PROGRAM MAIN
VAR
	fbBlinklicht : FB_Blinklicht;
	fbVereinzelung : FB_Vereinzelung;
	fbezylinder1 : FB_EZylinder;
	fbezylinder2 : FB_EZylinder;
	fbAmpel : FB_Ampel;
	fbTransport : FB_Transport;
	fbDispenser : FB_Dispenser;
	fbAbfuellmodul : FB_Abfuellmodul;
	fbManAchseX : FB_ManAchse;
	fbManAchseY : FB_ManAchse;
	fbManAchseZ : FB_ManAchse;
	ix : UINT;
	ry : REAL;
	ax : Axis_Ref;
END_VAR

ry := FUN_SCALE(TO_REAL(ix),4096,0,350,0);

	
fbAbfuellmodul(
	bEnable:= IFC_HW.bEnable, 
	bExecute:= IFC_HW.bExecute, 
	nstation:= , 
	bEinzelSens1:= IFC_HW.bEinzelSens1, 
	bEinzelSens2:= IFC_HW.bEinzelSens2, 
	bEinzelSens3:= IFC_HW.bEinzelSens3, 
	bEinzelSens4:= IFC_HW.bBandSens1, 
	bBandSens1:= IFC_HW.bBandSens1, 
	bBandSens2:= IFC_HW.bBandSens2, 
	bBandSens3:= IFC_HW.bBandSens3, 
	bBandSens4:= IFC_HW.bBandSens4, 
	bstopper1=> IFC_HW.bBandHub1, 
	bstopper2=> IFC_HW.bBandHub2, 
	bstopper3=>IFC_HW.bBandHub3, 
	estate=> , 
	bgate1=> fbeZylinder1.bgate, 
	bgate2=> fbeZylinder2.bgate, 
	axTransport:= IFC_HW.ax_BandMotor, 
	axDisp1:= IFC_HW.ax_Extruder1, 
	axDisp2:= IFC_HW.ax_Extruder2, 
	axDisp3:= IFC_HW.ax_Extruder3);
	
(*				
fbVereinzelung(
	benable:= IFC_HW.bEnable, 
	bexecute:= IFC_HW.bExecute, 
	bsensor1:= IFC_HW.bEinzelSens1, 
	bsensor2:= IFC_HW.bEinzelSens2, 
	bsensor3:= IFC_HW.bEinzelSens3, 
	bsensor4:= IFC_HW.bBandsens1, 
	bgate1=> fbeZylinder1.bgate, 
	bgate2=> fbeZylinder2.bgate, 
	estate=> );
	*)
	
	fbezylinder1(bgate:= , berror:= , bR1=>IFC_HW.bR1AKT1 , bR2=>IFC_HW.br2AKT1 );
	
	fbezylinder2(bgate:= , berror:= , bR1=>IFC_HW.bR1AKT2 , bR2=> IFC_HW.bR2AKT2);
	
	
	fbAmpel(estate:= fbAbfuellmodul.estate, bAmpelgruen=>IFC_HW.bAmpelGrun , bAmpelrot=>IFC_HW.bAmpelRot , bAmpelgelb=>IFC_HW.bAmpelGelb );
(*
fbTransport(
	bEnable:= IFC_Hw.bEnable, 
	bExecute:= IFC_HW.bExecute, 
	nstation:= 1, 
	bSens1:= IFC_HW.bBandSens1, 
	bSens2:= IFC_HW.bBandSens2, 
	bSens3:= IFC_HW.bBandSens3, 
	bSens4:= IFC_HW.bBandSens4, 
	eState=> , 
	bstopper1=> IFC_HW.bBandHub1, 
	bstopper2=> IFC_HW.bBandHub2, 
	bstopper3=> IFC_HW.bBandHub3, 
	ax:= IFC_HW.ax_BandMotor);

fbDispenser(
	benable:= IFC_Hw.bEnable, 
	bexecute:= IFC_HW.bExecute, 
	rVelocity:= 10, 
	rDistance:= 10, 
	estate=> , 
	ax:= IFC_HW.ax_Extruder1); *)
	
fbManAchseX(
	benable:= IFC_Hw.bEnable, 
	bexecute:= IFC_Hw.bExecute, 
	bEndschalter:= IFC_HW.bManEndXmin, 
	rPosition:= 150, 
	rVel:= 30, 
	estate=> , 
	ax:= IFC_HW.ax_ManX);

	
fbManAchseY(
	benable:= IFC_Hw.bEnable, 
	bexecute:= IFC_Hw.bExecute, 
	bEndschalter:= IFC_HW.bManEndYmin, 
	rPosition:= 150, 
	rVel:= 30, 
	estate=> , 
	ax:= IFC_HW.ax_ManY); 

fbManAchseZ(
	benable:= IFC_Hw.bEnable, 
	bexecute:= IFC_Hw.bExecute, 
	bEndschalter:= IFC_HW.bManEndZmin, 
	rPosition:= 150, 
	rVel:= 30, 
	estate=> , 
	ax:= IFC_HW.ax_ManZ);

END_PROGRAM

(* stored: Version 1.1.0.1, ProductVersion 3.1.4024.15
   POU MAIN: Id {bd947791-4b97-4a15-8e58-4d7bb5a41737}, SpecialFunc None *)
